KUKA KRL program: FlexPumpOn.src

&ACCESS RVO
&REL 1
&PARAM EDITMASK = *
&PARAM TEMPLATE = C:\KRC\Roboter\Template\vorgabe
DEF FlexPumpOn( )

;************************************************
;              CNC Robotics Ltd
;              www.cncrobotics.co.uk
;************************************************
;     Contact: helpdesk@cncrobotics.co.uk
;     Date: 25/09/23
;     Version: 0.9.46
;************************************************
; Description: Routine to turn off the Flex Pump
; 			   On
;************************************************

WAIT SEC 0
oTrackLubrication = TRUE

END
